// Mitsubishi GX Works2 project: e01   PLC: Q02/Q02H

PROGRAM MAIN
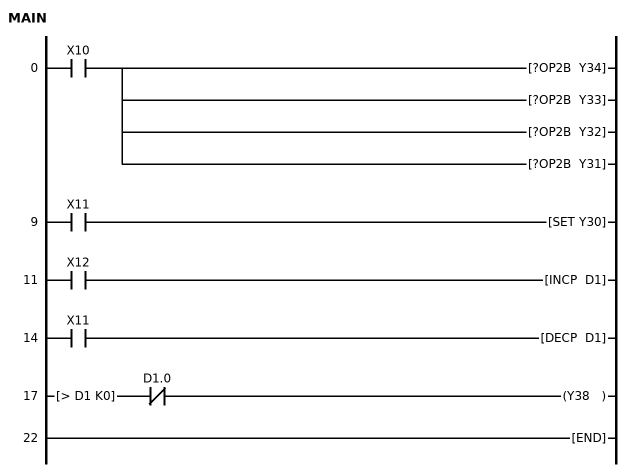
0     LD      X10
      ?OP2B   Y34
      ?OP2B   Y33
      ?OP2B   Y32
      ?OP2B   Y31
9     LD      X11
      SET     Y30
11    LD      X12
      INCP    D1
14    LD      X11
      DECP    D1
17    LD>     D1 K0
      ANI     D1.0
      OUT     Y38
22    END
END_PROGRAM
